Yaskawa INFORM job: X2_27-28(-50,-90).JBI

/JOB
//NAME X2_27-28(-50,-90)
//POS
///NPOS 352,352,352,16,0,0
///TOOL 0
///POSTYPE PULSE
///PULSE
C00000=-2348,-136985,-121477,-16,96092,-119
C00001=102627,-116827,-115343,23688,103226,-44542
C00002=115004,-86962,-92134,24001,100691,-40453
C00003=118842,-87386,-89376,23795,97842,-39618
C00004=120381,-87384,-88200,23717,96741,-39273
C00005=120377,-87274,-86494,23659,95829,-39457
C00006=120358,-87289,-86697,23665,95942,-39442
C00007=122537,-87238,-86673,23616,95334,-38762
C00008=120358,-87289,-86697,23665,95942,-39442
C00009=120413,-87366,-86683,23662,95882,-39433
C00010=120414,-83407,-84990,23721,96794,-39250
C00011=120413,-87366,-86683,23662,95882,-39433
C00012=118874,-87417,-87880,23731,96972,-39781
C00013=115033,-87126,-90695,23913,99792,-40627
C00014=115188,-84882,-91157,24044,101067,-40307
C00015=118973,-85347,-88418,23826,98226,-39491
C00016=120455,-85363,-87251,23745,97137,-39166
C00017=120452,-85286,-85558,23683,96217,-39352
C00018=120487,-85295,-85812,23691,96347,-39313
C00019=122635,-85238,-85785,23639,95749,-38643
C00020=120487,-85295,-85812,23691,96347,-39313
C00021=120483,-89746,-89095,23675,96102,-39363
C00022=120398,-93403,-88367,23560,93986,-39817
C00023=120400,-89378,-86736,23609,94965,-39621
C00024=120398,-93403,-88367,23560,93986,-39817
C00025=114754,-95185,-95401,23812,98729,-40947
C00026=113817,-96176,-94667,23309,84492,-38861
C00027=117813,-93582,-90807,22657,82424,-37804
C00028=119373,-92438,-89214,22393,81636,-37384
C00029=121634,-92435,-89210,21971,81030,-36673
C00030=120812,-92629,-89389,22126,81259,-36930
C00031=120809,-92377,-87626,22175,80372,-37096
C00032=120812,-92629,-89389,22126,81259,-36930
C00033=120909,-77641,-83091,21971,84792,-36245
C00034=120897,-73822,-81314,21956,85603,-36101
C00035=120909,-77641,-83091,21971,84792,-36245
C00036=115943,-80689,-88441,22878,87717,-37472
C00037=114304,-84462,-91699,24296,79100,-50020
C00038=117993,-82622,-88033,23316,76858,-49124
C00039=119438,-81769,-86512,22922,76000,-48762
C00040=121534,-81768,-86509,22277,75434,-48100
C00041=120893,-81605,-86471,22471,75662,-48293
C00042=120882,-79116,-84088,22491,75491,-48329
C00043=120893,-81605,-86471,22471,75662,-48293
C00044=120874,-97072,-87829,23296,69089,-49605
C00045=120882,-99825,-87797,23508,67765,-49878
C00046=120874,-97072,-87829,23296,69089,-49605
C00047=115137,-101258,-93439,24799,71949,-51221
C00048=121122,-106374,-107449,-1374,89824,-2285
C00049=126924,-83388,-91593,-24529,79629,49999
C00050=123244,-81641,-87969,-23551,77363,49118
C00051=121801,-80822,-86464,-23159,76497,48761
C00052=119718,-80838,-86473,-22519,75929,48107
C00053=120355,-80669,-86431,-22711,76157,48297
C00054=120355,-78205,-84050,-22728,75972,48332
C00055=120355,-80669,-86431,-22711,76157,48297
C00056=120389,-96242,-87887,-23521,69604,49623
C00057=120385,-99021,-87874,-23730,68282,49899
C00058=120389,-96242,-87887,-23521,69604,49623
C00059=126112,-100299,-93445,-25011,72503,51215
C00060=127424,-95125,-94496,-23537,84985,38865
C00061=123439,-92623,-90674,-22887,82890,37821
C00062=121881,-91514,-89094,-22623,82092,37406
C00063=119636,-91530,-89104,-22205,81483,36703
C00064=120453,-91715,-89278,-22359,81714,36957
C00065=120449,-91492,-87527,-22405,80819,37124
C00066=120453,-91715,-89278,-22359,81714,36957
C00067=120324,-76745,-82936,-22209,85198,36262
C00068=120328,-72933,-81149,-22194,85997,36116
C00069=120324,-76745,-82936,-22209,85198,36262
C00070=125282,-79685,-88237,-23118,88153,37475
C00071=126053,-84105,-90945,-24270,101400,40334
C00072=121317,-84665,-86997,-23961,97551,39378
C00073=120794,-84655,-86302,-23916,97014,39294
C00074=120791,-84616,-85408,-23898,96528,39392
C00075=120757,-84623,-85661,-23907,96658,39353
C00076=118619,-84583,-85646,-23856,96058,38687
C00077=120757,-84623,-85661,-23907,96658,39353
C00078=120851,-89642,-89189,-23884,96311,39457
C00079=120861,-92728,-88235,-23770,94318,39863
C00080=120850,-88708,-86596,-23821,95285,39665
C00081=120861,-92728,-88235,-23770,94318,39863
C00082=126087,-84100,-90943,-24271,101411,40344
C00083=126241,-86175,-91925,-24226,101032,40481
C00084=121422,-86671,-87791,-23936,97086,39512
C00085=120872,-86641,-86990,-23895,96491,39430
C00086=120871,-86598,-86346,-23873,96146,39499
C00087=120890,-86611,-86548,-23880,96260,39483
C00088=118722,-86577,-86536,-23832,95649,38808
C00089=120890,-86611,-86548,-23880,96260,39483
C00090=105063,-136064,-103329,-13656,63018,16453
C00091=105943,-129413,-101511,-13642,65401,16501
C00092=120836,-86689,-86535,-23876,96200,39475
C00093=126205,-86358,-90494,-24135,100129,40655
C00094=125851,-82973,-83923,-27955,66645,49280
C00095=122078,-79433,-79887,-26568,64829,48204
C00096=120947,-75344,-77359,-25987,64969,47712
C00097=120941,-87606,-78058,-27327,59684,49044
C00098=122175,-43746,-63261,-25567,94939,41852
C00099=109367,-31323,-61147,-11102,108854,34189
C00100=107960,-73866,-84355,-11763,95605,26787
C00101=120197,-78516,-82664,-23544,93398,30256
C00102=120674,-129805,-92807,-30414,50954,51524
C00103=120568,-142544,-87811,-37090,40465,55803
C00104=123719,-144899,-89705,-38330,41729,57027
C00105=131684,-150990,-93667,-41315,44633,60156
C00106=129569,-143343,-101170,-37382,56065,55166
C00107=120626,-84262,-98768,-23738,98439,36527
C00108=120626,-85138,-96217,-23600,96582,36901
C00109=120626,-85456,-94922,-23545,95698,37077
C00110=120469,-86348,-95216,-23512,95399,37081
C00111=120625,-86136,-87716,-24840,69295,42376
C00112=120625,-84905,-79807,-28619,54750,46053
C00113=120674,-84200,-73221,-29616,52346,46820
C00114=120694,-85495,-80856,-24885,69158,42438
C00115=120625,-86085,-86255,-23338,89936,38209
C00116=120426,-89896,-87913,-23311,89017,38317
C00117=120625,-86141,-87502,-23348,90617,38076
C00118=120625,-86117,-90396,-23390,92270,37753
C00119=121122,-106374,-107449,-1374,89824,-2285
C00120=115389,-83619,-83840,27729,66202,-49282
C00121=119161,-80016,-79774,26335,64406,-48194
C00122=120546,-78290,-78340,25753,63980,-47732
C00123=118816,-53732,-67922,25413,88359,-43218
C00124=120555,-20800,-48886,25341,110394,-38056
C00125=120540,-55987,-71055,24625,106356,-38968
C00126=122541,-110534,-92373,22580,69456,-43286
C00127=118405,-143902,-85879,49364,33417,-58427
C00128=117619,-149172,-81328,56749,30391,-62419
C00129=116407,-166632,-89102,63406,28902,-66105
C00130=115676,-54235,-75024,25023,110799,-39825
C00131=118805,-64147,-80292,27733,101935,-40879
C00132=120626,-85310,-99014,23481,98015,-36524
C00133=120626,-86187,-96453,23350,96148,-36894
C00134=120608,-87043,-95140,23285,95004,-37126
C00135=120561,-87834,-95469,23281,94829,-37179
C00136=120625,-86662,-87587,24592,68893,-42354
C00137=120624,-85616,-79792,28395,54313,-46043
C00138=120594,-85215,-73113,29470,51713,-46859
C00139=120625,-86330,-81078,24616,68777,-42377
C00140=119608,-72473,-79941,24560,98029,-43290
C00141=120456,-60135,-73698,25012,105696,-48505
C00142=120625,-87037,-87669,23119,90208,-38053
C00143=120626,-87011,-90570,23155,91868,-37731
C00144=120666,-77011,-108669,24508,106824,-34682
C00145=120666,-77011,-108669,24508,106824,-34682
C00146=69969,-70044,-127853,-26190,66176,42607
C00147=164066,-57873,-122395,-24689,68505,41679
C00148=164066,-57873,-122395,-24689,68505,41679
C00149=160176,-49519,-119791,-24551,119921,39872
C00150=160176,-63483,-121326,-22850,113002,41438
C00151=158640,-65340,-120741,-22195,111473,41297
C00152=158591,-68589,-120293,-21868,109653,41643
C00153=157443,-69457,-121106,-21570,109470,41332
C00154=156525,-70687,-121652,-21280,109008,41144
C00155=157421,-68776,-121134,-21620,109807,41260
C00156=165312,-86424,-128504,-22962,107296,44197
C00157=165830,-86354,-127308,-22986,106767,44469
C00158=165199,-83493,-126223,-22948,107364,44147
C00159=166594,-89849,-128602,-23030,106020,44865
C00160=164066,-57873,-122395,-24689,117052,41679
C00161=137183,-48540,-113103,-27062,110870,33097
C00162=133437,-50146,-110771,-25387,107987,32705
C00163=131981,-50551,-109735,-24766,106894,32528
C00164=131972,-53362,-109280,-24521,105318,32870
C00165=131636,-52132,-109559,-24518,105977,32629
C00166=130703,-53161,-109590,-24138,105304,32500
C00167=129879,-53398,-109717,-23857,105082,32305
C00168=131928,-52773,-109383,-24556,105642,32786
C00169=129764,-110950,-131053,-20350,81074,33499
C00170=129689,-122862,-131886,-20674,75787,34382
C00171=129370,-114001,-129067,-20345,78360,33827
C00172=129689,-122862,-131886,-20674,75787,34382
C00173=132778,-100905,-131254,-21387,86712,33498
C00174=143318,-75184,-130722,-7426,108145,5953
C00175=142042,-70835,-125479,-6985,107076,5675
C00176=141569,-69161,-123389,-6821,106623,5573
C00177=141558,-72780,-123049,-6738,104567,5686
C00178=141593,-72294,-123187,-6761,104902,5677
C00179=140967,-66354,-120569,-6623,106293,5428
C00180=141593,-72294,-123187,-6761,104902,5677
C00181=143345,-79213,-130741,-7340,106105,6087
C00182=143299,-74412,-130544,-7434,108429,5930
C00183=142026,-70178,-125329,-6991,107319,5656
C00184=141554,-68541,-123249,-6826,106852,5556
C00185=141544,-72173,-122918,-6742,104795,5669
C00186=141535,-71558,-123086,-6755,105212,5644
C00187=140912,-65651,-120469,-6618,106588,5397
C00188=141535,-71558,-123086,-6755,105212,5644
C00189=143280,-78289,-130595,-7337,106482,6046
C00190=143232,-73654,-130370,-7428,108704,5895
C00191=141965,-69530,-125182,-6983,107555,5626
C00192=141496,-67928,-123110,-6817,107076,5527
C00193=141485,-71574,-122787,-6732,105017,5641
C00194=141522,-70879,-122980,-6762,105492,5624
C00195=140900,-65004,-120364,-6625,106853,5379
C00196=141522,-70879,-122980,-6762,105492,5624
C00197=143263,-77436,-130447,-7347,106826,6020
C00198=97122,-37708,-107994,29413,114613,-34215
C00199=100765,-40257,-106178,27624,111617,-33971
C00200=102190,-41052,-105346,26964,110463,-33848
C00201=102184,-43828,-104954,26656,108968,-34218
C00202=102229,-43254,-105047,26705,109274,-34130
C00203=104151,-44223,-105589,26045,108681,-33706
C00204=102229,-43254,-105047,26705,109274,-34130
C00205=102390,-95092,-126215,23236,87986,-35228
C00206=102126,-106454,-127212,23433,83236,-36243
C00207=102723,-99043,-124596,23148,85111,-35678
C00208=102126,-106454,-127212,23433,83236,-36243
C00209=98351,-76946,-122874,24964,95636,-34932
C00210=98001,-57475,-123101,17996,113820,-36592
C00211=101536,-60773,-120906,16470,110382,-36160
C00212=102910,-63141,-119733,15828,108317,-36071
C00213=102916,-65026,-119479,15713,107233,-36217
C00214=102928,-64308,-119579,15751,107645,-36158
C00215=105169,-65555,-120144,15037,107042,-35610
C00216=102928,-64308,-119579,15751,107645,-36158
C00217=100368,-93898,-131351,15864,100368,-37874
C00218=97661,-87630,-128580,16731,102276,-38427
C00219=97996,-84252,-127310,16710,103135,-38207
C00220=97637,-87591,-128732,16747,102389,-38418
C00221=98001,-57475,-123101,17996,113820,-36592
C00222=99672,-7498,-88471,25376,120102,-35641
C00223=102088,-13346,-89114,23936,117260,-35660
C00224=103047,-14853,-89113,23458,116364,-35598
C00225=103070,-15280,-89318,23419,116275,-35613
C00226=103053,-14956,-89343,23464,116445,-35580
C00227=111428,-26181,-98637,10737,112296,-30408
C00228=102060,-12538,-89166,24052,117675,-35572
C00229=99645,-6651,-88487,25511,120511,-35544
C00230=110953,-13508,-91662,10573,109125,24437
C00231=110055,-18058,-91129,10746,106581,23991
C00232=118115,-24092,-94041,-1176,104714,22608
C00233=109847,-18561,-90498,10785,105963,23883
C00234=111445,-19708,-91242,10156,105696,24257
C00235=118682,-20843,-91970,7294,105023,25985
C00236=108853,-8664,-84384,24098,112429,23291
C00237=120831,-18883,-92219,6481,106051,26563
C00238=108247,-47697,-110693,11257,103619,23266
C00239=108001,-45758,-107370,11293,102615,23108
C00240=93743,-22704,-93084,31932,116237,9910
C00241=103043,-28379,-96833,28832,113378,11880
C00242=99567,-22662,-96038,30605,116358,11712
C00243=121744,-14004,-92551,6221,108699,26920
C00244=120102,-53038,-115079,-8947,92663,44391
C00245=120610,-122376,-128753,-45788,73253,81068
C00246=120610,-123649,-126232,-46257,71693,81820
C00247=114942,-121659,-128592,-38094,72140,80087
C00248=110746,-115512,-128718,-32121,74014,77680
C00249=111140,-116612,-128713,-32226,73312,78150
C00250=112123,-116971,-127920,-32543,72557,78927
C00251=114439,-125713,-130131,-33559,69229,81351
C00252=117557,-125023,-128034,-34922,66197,84237
C00253=123831,-113405,-131509,-37414,82436,80766
C00254=120611,-116611,-133297,-36284,80720,80097
C00255=120611,-116611,-133297,-36284,54343,80097
C00256=99428,-107843,-133398,6584,68498,81557
C00257=78879,-54177,-103402,55937,89044,85268
C00258=78429,-99723,-127104,45672,96643,84222
C00259=82364,-110385,-127773,44232,91185,83459
C00260=83904,-116944,-128983,43779,88549,82984
C00261=84962,-116458,-129077,42971,88317,83920
C00262=85753,-115873,-128369,42851,86976,84102
C00263=94278,-102678,-129331,33632,95313,84379
C00264=94252,-98051,-127422,33733,96332,84676
C00265=92227,-97102,-128188,34391,97842,84417
C00266=83296,-105916,-131418,40048,95342,83077
C00267=112976,-81346,-133029,11053,104292,84731
C00268=138914,-76030,-130615,-14013,102422,84743
C00269=139405,-82424,-128484,-14961,97637,85019
C00270=139610,-84860,-127656,-14962,95960,85285
C00271=122825,-93017,-130267,6502,91067,84006
C00272=122185,-92165,-130257,6747,91537,83850
C00273=122216,-90116,-129760,6745,92278,83897
C00274=121098,-81728,-131688,7259,97815,83901
C00275=117564,-73996,-132555,6245,103794,67045
C00276=120619,-75058,-128623,-5257,106122,114
C00277=120619,-82255,-128190,-5150,102172,284
C00278=120619,-84669,-127718,-5117,100646,349
C00279=112025,-83330,-127195,-2462,100682,-2074
C00280=125410,-84211,-127707,-6591,101158,1679
C00281=116389,-83882,-127652,-3819,100819,-855
C00282=120619,-81538,-128040,-5156,102448,272
C00283=120619,-74311,-128456,-5266,106402,102
C00284=120619,-74726,-128566,4732,106271,-192
C00285=120619,-81960,-128145,4635,102308,-346
C00286=120619,-84896,-127978,4605,100704,-408
C00287=130171,-82621,-126955,1656,100942,2285
C00288=124481,-84935,-127680,3411,100342,674
C00289=124544,-84819,-127737,3393,100431,696
C00290=120619,-82679,-128294,4629,102031,-356
C00291=132569,-75475,-129249,4725,105990,-203
C00292=136339,-73848,-128583,3524,106271,812
C00293=115610,-90997,-132796,9664,98154,47330
C00294=101030,-93647,-129382,39129,95529,59479
C00295=126122,-118259,-133558,37742,75798,85079
C00296=126123,-123502,-128947,38676,71399,83468
C00297=126367,-125496,-128832,38806,70431,83204
C00298=126259,-125638,-129343,38123,70704,84047
C00299=126452,-122750,-128309,37875,71302,84347
C00300=126394,-120456,-127460,37773,71850,84523
C00301=124054,-126150,-130879,35007,72357,80836
C00302=128390,-137176,-133704,31743,64167,79569
C00303=127393,-110720,-125425,30503,71855,81401
C00304=124670,-119490,-131862,32313,77272,81796
C00305=123468,-105545,-131306,32649,85926,83785
C00306=123468,-105545,-131306,32649,65045,83785
C00307=138629,-76986,-116006,-44057,63514,71452
C00308=138629,-76986,-116006,-43820,94287,71434
C00309=134687,-82864,-115400,-42250,90109,71636
C00310=135664,-119265,-122373,-47079,71549,79745
C00311=132914,-91853,-117066,-41458,84473,72364
C00312=132788,-89730,-116313,-41385,84897,72145
C00313=132694,-88516,-115506,-41345,84954,72084
C00314=132043,-80417,-112459,-40576,87939,70586
C00315=130204,-77793,-113758,-38013,92059,70441
C00316=128524,-79115,-118595,-35047,97544,70713
C00317=132051,-72530,-119355,-36693,101910,70485
C00318=103939,-76664,-132684,-5369,102917,72052
C00319=89328,-90531,-135287,12506,96574,73027
C00320=80068,-79251,-126452,22073,101797,73002
C00321=79731,-82396,-126595,22049,100450,72647
C00322=75389,-93321,-128367,26734,94516,71144
C00323=89823,-118490,-137568,8328,79761,70288
C00324=89823,-118490,-137568,8328,79761,70288
C00325=89554,-115143,-136518,8419,80849,70278
C00326=90481,-87040,-133249,3898,95478,71874
C00327=121995,-40580,-113920,-16331,113160,53817
C00328=134131,-13261,-91828,-23304,117904,34003
C00329=134130,-17922,-91482,-22725,115495,34532
C00330=134178,-18161,-90930,-22645,115075,34636
C00331=134130,-19018,-91366,-22584,114907,34660
C00332=134135,-19080,-91406,-22584,114899,34666
C00333=130040,-16797,-91734,-17058,116519,30349
C00334=134130,-17121,-91555,-22821,115917,34441
C00335=134485,-13609,-94717,-23816,119438,33744
C00336=134125,-15266,-91655,-12564,108610,-23590
C00337=134126,-19967,-91222,-12356,105989,-23311
C00338=128619,-18785,-91351,-4606,108870,-22773
C00339=134001,-21196,-91423,-12272,105476,-23287
C00340=133837,-21232,-91027,-12191,105205,-23306
C00341=133810,-21099,-91074,-12188,105299,-23320
C00342=142675,1303,-75956,-28153,117136,-18516
C00343=136270,-18169,-92488,-13326,107877,-22987
C00344=160414,-17591,-92076,-34517,119430,-9586
C00345=156591,-5353,-82577,-31368,124461,-10572
C00346=145789,-11555,-87834,-25790,123238,-6673
C00347=150771,-16897,-91755,-28044,119951,-5168
C00348=137962,-9823,-90715,-14308,111174,-22977
C00349=135096,-37202,-106359,-15392,53710,-23809
C00350=91634,-70237,-111781,-11635,26322,-15777
C00351=-2394,-140510,-122466,-18,94889,-134
BC00000=133244,518772,1075139
BC00001=133244,374008,1075139
BC00002=133244,374008,1075139
BC00003=133244,374008,1075139
BC00004=133244,374008,1075139
BC00005=133244,374008,1075139
BC00006=133244,374008,1075139
BC00007=133244,374008,1075139
BC00008=133244,374008,1075139
BC00009=133244,374008,1075139
BC00010=133244,374008,1075139
BC00011=133244,374008,1075139
BC00012=133244,374008,1075139
BC00013=133244,374008,1075139
BC00014=133336,405551,1075139
BC00015=133336,405551,1075139
BC00016=133336,405551,1075139
BC00017=133336,405551,1075139
BC00018=133336,405551,1075139
BC00019=133336,405551,1075139
BC00020=133336,405551,1075139
BC00021=133336,405551,1075139
BC00022=133336,405551,1075139
BC00023=133336,405551,1075139
BC00024=133336,405551,1075139
BC00025=133336,405551,1075139
BC00026=104477,408619,1075139
BC00027=104477,408619,1075139
BC00028=104477,408619,1075139
BC00029=104477,408619,1075139
BC00030=104477,408619,1075139
BC00031=104477,408619,1075139
BC00032=104477,408619,1075139
BC00033=104477,408619,1075139
BC00034=104477,408619,1075139
BC00035=104477,408619,1075139
BC00036=104477,408619,1075139
BC00037=104582,411051,1075139
BC00038=104582,411051,1075139
BC00039=104582,411051,1075139
BC00040=104582,411051,1075139
BC00041=104582,411051,1075139
BC00042=104582,411051,1075139
BC00043=104582,411051,1075139
BC00044=104582,411051,1075139
BC00045=104582,411051,1075139
BC00046=104582,411051,1075139
BC00047=104582,411051,1075139
BC00048=209905,391148,1075139
BC00049=330495,411073,1075139
BC00050=330495,411073,1075139
BC00051=330495,411073,1075139
BC00052=330495,411073,1075139
BC00053=330495,411073,1075139
BC00054=330495,411073,1075139
BC00055=330495,411073,1075139
BC00056=330495,411073,1075139
BC00057=330495,411073,1075139
BC00058=330495,411073,1075139
BC00059=330495,411073,1075139
BC00060=330336,408559,1075139
BC00061=330336,408559,1075139
BC00062=330336,408559,1075139
BC00063=330336,408559,1075139
BC00064=330336,408559,1075139
BC00065=330336,408559,1075139
BC00066=330336,408559,1075139
BC00067=330336,408559,1075139
BC00068=330336,408559,1075139
BC00069=330336,408559,1075139
BC00070=330336,408559,1075139
BC00071=301636,405299,1075139
BC00072=301637,405300,1075138
BC00073=301637,405300,1075137
BC00074=301636,405299,1075139
BC00075=301636,405299,1075139
BC00076=301636,405299,1075139
BC00077=301636,405299,1075139
BC00078=301636,405299,1075139
BC00079=301636,405299,1075139
BC00080=301636,405299,1075139
BC00081=301636,405299,1075139
BC00082=301636,405299,1075139
BC00083=301924,373758,1075139
BC00084=301924,373758,1075139
BC00085=301924,373758,1075139
BC00086=301924,373758,1075139
BC00087=301924,373758,1075139
BC00088=301924,373758,1075139
BC00089=301924,373758,1075139
BC00090=301924,373758,1075139
BC00091=301924,373758,1075139
BC00092=301924,373758,1075139
BC00093=301924,373758,1075139
BC00094=304905,422275,1075139
BC00095=304905,422275,1075139
BC00096=304905,422275,1075139
BC00097=304905,422275,1075139
BC00098=304905,422275,1075139
BC00099=304905,422275,1075139
BC00100=304905,422275,1075139
BC00101=304905,422275,1075139
BC00102=304905,422275,1075139
BC00103=304905,422275,1075139
BC00104=304905,422275,1075139
BC00105=304905,422275,1075139
BC00106=308182,411224,1075150
BC00107=321948,364809,1075193
BC00108=327549,363919,1075193
BC00109=329789,363562,1075193
BC00110=329784,365099,1075193
BC00111=329679,406352,1075193
BC00112=329645,424796,1075193
BC00113=329621,438429,1075193
BC00114=329656,420343,1075193
BC00115=329731,391181,1075193
BC00116=329680,407690,1075193
BC00117=327439,408070,1075193
BC00118=321838,409018,1075193
BC00119=209905,391148,1075139
BC00120=130051,422412,1075139
BC00121=130051,422412,1075139
BC00122=130051,422412,1075139
BC00123=130051,422412,1075139
BC00124=130051,422412,1075139
BC00125=130051,422412,1075139
BC00126=130051,422412,1075139
BC00127=130051,422412,1075139
BC00128=130052,422412,1075139
BC00129=130051,422412,1075139
BC00130=130051,422412,1075139
BC00131=129375,420117,1075141
BC00132=113133,364939,1075193
BC00133=107556,364016,1075193
BC00134=105325,363648,1075192
BC00135=105320,365183,1075193
BC00136=105215,406346,1075193
BC00137=105181,424701,1075193
BC00138=105157,438341,1075193
BC00139=105192,420360,1075193
BC00140=105266,391265,1075193
BC00141=105215,407774,1075193
BC00142=107446,408166,1075193
BC00143=113024,409146,1075193
BC00144=113024,409146,1075193
BC00145=113024,615302,1075193
BC00146=61085,522072,1075139
BC00147=61085,522072,1075139
BC00148=61085,344205,1075139
BC00149=61085,344205,1072934
BC00150=61085,344205,1075139
BC00151=61085,344205,1075139
BC00152=61085,344205,1075139
BC00153=61085,344205,1075139
BC00154=61085,344205,1075139
BC00155=61085,344205,1075139
BC00156=61085,344205,1075139
BC00157=61085,344205,1075139
BC00158=61085,344205,1075139
BC00159=61085,344205,1075139
BC00160=61085,344205,1075139
BC00161=23280,347448,1075139
BC00162=23280,347448,1075139
BC00163=23280,347448,1075139
BC00164=23280,347448,1075139
BC00165=23280,347448,1075139
BC00166=23280,347448,1075139
BC00167=23280,347448,1075139
BC00168=23280,347448,1075139
BC00169=23280,347448,1075139
BC00170=23280,347448,1075139
BC00171=23280,347448,1075139
BC00172=23280,347448,1075139
BC00173=23280,347448,1075139
BC00174=188977,346610,1075139
BC00175=188977,346610,1075139
BC00176=188977,346610,1075139
BC00177=188977,346610,1075139
BC00178=188977,346610,1075139
BC00179=188977,346610,1075139
BC00180=188977,346610,1075139
BC00181=188977,346610,1075139
BC00182=244494,346740,1075139
BC00183=244494,346740,1075139
BC00184=244494,346740,1075139
BC00185=244494,346740,1075139
BC00186=244494,346740,1075139
BC00187=244494,346740,1075139
BC00188=244494,346740,1075139
BC00189=244494,346740,1075139
BC00190=299376,346854,1075139
BC00191=299376,346854,1075139
BC00192=299376,346854,1075139
BC00193=299376,346854,1075139
BC00194=299376,346854,1075139
BC00195=299376,346854,1075139
BC00196=299376,346854,1075139
BC00197=299376,346854,1075139
BC00198=398158,351394,1075139
BC00199=398158,351394,1075139
BC00200=398158,351394,1075139
BC00201=398158,351394,1075139
BC00202=398158,351394,1075139
BC00203=398158,351394,1075139
BC00204=398158,351394,1075139
BC00205=398158,351394,1075139
BC00206=398158,351394,1075139
BC00207=398158,351394,1075139
BC00208=398158,351394,1075139
BC00209=398158,351394,1075139
BC00210=398158,355332,1075139
BC00211=398158,355332,1075139
BC00212=398158,355332,1075139
BC00213=398158,355332,1075139
BC00214=398158,355332,1075139
BC00215=398158,355332,1075139
BC00216=398158,355332,1075139
BC00217=398158,355332,1075139
BC00218=398158,355332,1075139
BC00219=398158,355332,1075139
BC00220=398158,355332,1075139
BC00221=398158,355332,1075139
BC00222=398158,400322,1075139
BC00223=398158,397462,1075139
BC00224=398158,396318,1075139
BC00225=398158,391714,1075139
BC00226=398158,377425,1075139
BC00227=398158,372820,1075139
BC00228=398158,373964,1075139
BC00229=398158,376823,1075139
BC00230=398158,418089,1075139
BC00231=398158,413055,1075139
BC00232=398158,411041,1075139
BC00233=398158,411041,1075139
BC00234=398158,407701,1075139
BC00235=398158,394074,1075139
BC00236=398157,390799,1075138
BC00237=398158,392757,1075139
BC00238=398158,392757,1075139
BC00239=398158,392757,1075139
BC00240=398158,392757,1075139
BC00241=398158,392757,1075139
BC00242=398158,392757,1075139
BC00243=398158,397791,1075139
BC00244=368036,376425,1075139
BC00245=305380,328053,1075139
BC00246=311014,327368,1075139
BC00247=313268,327093,1075139
BC00248=314020,306251,1075134
BC00249=314937,305830,1075134
BC00250=316315,305197,1075135
BC00251=320257,303387,1075136
BC00252=325137,301146,1075137
BC00253=323904,301076,1075139
BC00254=319263,301619,1075139
BC00255=319263,301619,1075139
BC00256=354630,317867,1075139
BC00257=398158,344123,1075139
BC00258=398158,328829,1075139
BC00259=398158,328117,1075139
BC00260=398158,327832,1075139
BC00261=398158,306302,1075139
BC00262=398158,307654,1075139
BC00263=398158,299863,1075139
BC00264=398158,299863,1075139
BC00265=398158,299850,1075139
BC00266=398158,299818,1075139
BC00267=398158,306594,1075139
BC00268=398158,312941,1075139
BC00269=398158,312327,1075139
BC00270=398158,311910,1075139
BC00271=398158,311948,1075139
BC00272=398158,311948,1075139
BC00273=398158,311948,1075139
BC00274=398158,312262,1075139
BC00275=361275,323313,1075139
BC00276=206057,349327,1075139
BC00277=206787,343889,1075139
BC00278=207078,341714,1075139
BC00279=207078,341714,1075139
BC00280=265248,341851,1075139
BC00281=265248,341851,1075139
BC00282=264956,344026,1075139
BC00283=264226,349464,1075139
BC00284=226795,349421,1075139
BC00285=226137,343980,1075139
BC00286=225873,341804,1075139
BC00287=225873,341804,1075139
BC00288=182394,341701,1075139
BC00289=167704,341666,1075139
BC00290=167967,343843,1075139
BC00291=168625,349284,1075139
BC00292=168625,349284,1075139
BC00293=110827,349284,1075139
BC00294=117018,341898,1075139
BC00295=129083,327506,1075139
BC00296=123497,326795,1075139
BC00297=121263,326510,1075139
BC00298=120594,305154,1075139
BC00299=120594,305154,1075139
BC00300=120594,305154,1075139
BC00301=111835,301464,1075139
BC00302=111835,301467,1075137
BC00303=111835,301467,1075137
BC00304=111094,300785,1075138
BC00305=115319,301016,1075139
BC00306=115319,315076,1075139
BC00307=1592,364988,1075139
BC00308=1592,342862,1075139
BC00309=1592,342176,1075139
BC00310=1592,341902,1075139
BC00311=1592,321468,1075139
BC00312=1592,321468,1075139
BC00313=1592,321468,1075139
BC00314=1592,322137,1075139
BC00315=1592,315667,1075139
BC00316=1592,307060,1075139
BC00317=1592,307005,1075139
BC00318=5534,309480,1075139
BC00319=11068,305519,1075139
BC00320=9993,304471,1075139
BC00321=9607,304094,1075139
BC00322=9607,304094,1075139
BC00323=9607,304094,1075139
BC00324=9607,304094,1075139
BC00325=9607,304094,1075139
BC00326=1592,304326,1075139
BC00327=7124,350617,1075139
BC00328=20477,398593,1075139
BC00329=25318,395756,1075139
BC00330=27254,394622,1075139
BC00331=27284,390018,1075139
BC00332=27318,375728,1075139
BC00333=27313,372783,1075139
BC00334=25374,372258,1075139
BC00335=20533,375095,1075139
BC00336=41909,417655,1075139
BC00337=40292,412613,1075139
BC00338=39645,410596,1075139
BC00339=39645,410596,1075139
BC00340=42951,407272,1075139
BC00341=56475,393709,1075139
BC00342=56475,393709,1075139
BC00343=60436,392410,1075139
BC00344=60436,392410,1075139
BC00345=60435,392411,1075136
BC00346=60435,392411,1075136
BC00347=60435,392411,1075136
BC00348=62053,397452,1075139
BC00349=63646,397452,1075139
BC00350=86333,436115,1075139
BC00351=134837,518772,1075139
EC00000=443420,372643
EC00001=443420,372643
EC00002=443420,372643
EC00003=443420,372643
EC00004=443420,372643
EC00005=443420,372643
EC00006=443420,372643
EC00007=443420,372643
EC00008=443420,372643
EC00009=443420,372643
EC00010=443420,372643
EC00011=443420,372643
EC00012=443420,372643
EC00013=443420,372643
EC00014=443420,372643
EC00015=443420,372643
EC00016=443420,372643
EC00017=443420,372643
EC00018=443420,372643
EC00019=443420,372643
EC00020=443420,372643
EC00021=443420,372643
EC00022=443420,372643
EC00023=443420,372643
EC00024=443420,372643
EC00025=443420,372643
EC00026=443420,372643
EC00027=443420,372643
EC00028=443420,372643
EC00029=443420,372643
EC00030=443420,372643
EC00031=443420,372643
EC00032=443420,372643
EC00033=443420,372643
EC00034=443420,372643
EC00035=443420,372643
EC00036=443420,372643
EC00037=443420,372643
EC00038=443420,372643
EC00039=443420,372643
EC00040=443420,372643
EC00041=443420,372643
EC00042=443420,372643
EC00043=443420,372643
EC00044=443420,372643
EC00045=443420,372643
EC00046=443420,372643
EC00047=443420,372643
EC00048=443420,372643
EC00049=443420,372643
EC00050=443420,372643
EC00051=443420,372643
EC00052=443420,372643
EC00053=443420,372643
EC00054=443420,372643
EC00055=443420,372643
EC00056=443420,372643
EC00057=443420,372643
EC00058=443420,372643
EC00059=443420,372643
EC00060=443420,372643
EC00061=443420,372643
EC00062=443420,372643
EC00063=443420,372643
EC00064=443420,372643
EC00065=443420,372643
EC00066=443420,372643
EC00067=443420,372643
EC00068=443420,372643
EC00069=443420,372643
EC00070=443420,372643
EC00071=443420,372643
EC00072=443419,372644
EC00073=443418,372644
EC00074=443420,372643
EC00075=443420,372643
EC00076=443420,372643
EC00077=443420,372643
EC00078=443420,372643
EC00079=443420,372643
EC00080=443420,372643
EC00081=443420,372643
EC00082=443420,372643
EC00083=443420,372643
EC00084=443420,372643
EC00085=443420,372643
EC00086=443420,372643
EC00087=443420,372643
EC00088=443420,372643
EC00089=443420,372643
EC00090=443420,372643
EC00091=443420,372643
EC00092=443420,372643
EC00093=443420,372643
EC00094=443420,372643
EC00095=443420,372643
EC00096=443420,372643
EC00097=443420,372643
EC00098=443420,372643
EC00099=443420,372643
EC00100=443420,372643
EC00101=443420,372643
EC00102=443420,372643
EC00103=443420,372643
EC00104=443420,372643
EC00105=443420,372643
EC00106=443420,372643
EC00107=443420,372643
EC00108=443420,372643
EC00109=443420,372643
EC00110=443420,372643
EC00111=443420,372643
EC00112=443420,372643
EC00113=443420,372643
EC00114=443420,372643
EC00115=443420,372643
EC00116=443420,372643
EC00117=443420,372643
EC00118=443420,372643
EC00119=443420,372643
EC00120=443420,372643
EC00121=443420,372643
EC00122=443420,372643
EC00123=443420,372643
EC00124=443420,372643
EC00125=443420,372643
EC00126=443420,372643
EC00127=443420,372643
EC00128=443419,372642
EC00129=443420,372643
EC00130=443420,372643
EC00131=443420,372643
EC00132=443420,372643
EC00133=443420,372643
EC00134=443419,372643
EC00135=443420,372643
EC00136=443420,372643
EC00137=443420,372643
EC00138=443420,372643
EC00139=443420,372643
EC00140=443420,372643
EC00141=443420,372643
EC00142=443420,372643
EC00143=443420,372643
EC00144=443420,372643
EC00145=443420,372643
EC00146=798156,372643
EC00147=798156,372643
EC00148=798156,372643
EC00149=798156,372643
EC00150=798156,372643
EC00151=798156,372643
EC00152=798156,372643
EC00153=798156,372643
EC00154=798156,372643
EC00155=798156,372643
EC00156=798156,372643
EC00157=798156,372643
EC00158=798156,372643
EC00159=798156,372643
EC00160=798156,372643
EC00161=798156,372643
EC00162=798156,372643
EC00163=798156,372643
EC00164=798156,372643
EC00165=798156,372643
EC00166=798156,372643
EC00167=798156,372643
EC00168=798156,372643
EC00169=798156,372643
EC00170=798156,372643
EC00171=798156,372643
EC00172=798156,372643
EC00173=798156,372643
EC00174=798156,372643
EC00175=798156,372643
EC00176=798156,372643
EC00177=798156,372643
EC00178=798156,372643
EC00179=798156,372643
EC00180=798156,372643
EC00181=798156,372643
EC00182=798156,372643
EC00183=798156,372643
EC00184=798156,372643
EC00185=798156,372643
EC00186=798156,372643
EC00187=798156,372643
EC00188=798156,372643
EC00189=798156,372643
EC00190=798156,372643
EC00191=798156,372643
EC00192=798156,372643
EC00193=798156,372643
EC00194=798156,372643
EC00195=798156,372643
EC00196=798156,372643
EC00197=798156,372643
EC00198=798156,372643
EC00199=798156,372643
EC00200=798156,372643
EC00201=798156,372643
EC00202=798156,372643
EC00203=798156,372643
EC00204=798156,372643
EC00205=798156,372643
EC00206=798156,372643
EC00207=798156,372643
EC00208=798156,372643
EC00209=798156,372643
EC00210=798156,372643
EC00211=798156,372643
EC00212=798156,372643
EC00213=798156,372643
EC00214=798156,372643
EC00215=798156,372643
EC00216=798156,372643
EC00217=798156,372643
EC00218=798156,372643
EC00219=798156,372643
EC00220=798156,372643
EC00221=798156,372643
EC00222=798156,372643
EC00223=798156,372643
EC00224=798156,372643
EC00225=798156,372643
EC00226=798156,372643
EC00227=798156,372643
EC00228=798156,372643
EC00229=798156,372643
EC00230=798156,372643
EC00231=798156,372643
EC00232=798156,372643
EC00233=798156,372643
EC00234=798156,372643
EC00235=798156,372643
EC00236=798153,372643
EC00237=798156,372643
EC00238=798156,372643
EC00239=798156,372643
EC00240=798156,372643
EC00241=798156,372643
EC00242=798156,372643
EC00243=798156,372643
EC00244=798156,372643
EC00245=798156,372643
EC00246=798156,372643
EC00247=798156,372643
EC00248=798154,372643
EC00249=798154,372643
EC00250=798155,372644
EC00251=798155,372644
EC00252=798155,372643
EC00253=798156,372643
EC00254=798156,372643
EC00255=798156,372643
EC00256=798156,372643
EC00257=798156,372643
EC00258=798156,372643
EC00259=798156,372643
EC00260=798156,372643
EC00261=798156,372643
EC00262=798156,372643
EC00263=798156,372643
EC00264=798156,372643
EC00265=798156,372643
EC00266=798156,372643
EC00267=798156,372643
EC00268=798156,372643
EC00269=798156,372643
EC00270=798156,372643
EC00271=798156,372643
EC00272=798156,372643
EC00273=798156,372643
EC00274=798156,372643
EC00275=798156,372643
EC00276=798156,372643
EC00277=798156,372643
EC00278=798156,372643
EC00279=798156,372643
EC00280=798156,372643
EC00281=798156,372643
EC00282=798156,372643
EC00283=798156,372643
EC00284=798156,372643
EC00285=798156,372643
EC00286=798156,372643
EC00287=798156,372643
EC00288=798156,372643
EC00289=798156,372643
EC00290=798156,372643
EC00291=798156,372643
EC00292=798156,372643
EC00293=798156,372643
EC00294=798156,372643
EC00295=798156,372643
EC00296=798156,372643
EC00297=798156,372643
EC00298=798156,372643
EC00299=798156,372643
EC00300=798156,372643
EC00301=798156,372643
EC00302=798155,372643
EC00303=798155,372643
EC00304=798156,372643
EC00305=798156,372643
EC00306=798156,372643
EC00307=798156,372643
EC00308=798156,372643
EC00309=798156,372643
EC00310=798156,372643
EC00311=798156,372643
EC00312=798156,372643
EC00313=798156,372643
EC00314=798156,372643
EC00315=798156,372643
EC00316=798156,372643
EC00317=798156,372643
EC00318=798156,372643
EC00319=798156,372643
EC00320=798156,372643
EC00321=798156,372643
EC00322=798156,372643
EC00323=798156,372643
EC00324=798156,372643
EC00325=798156,372643
EC00326=798156,372643
EC00327=798156,372643
EC00328=798156,372643
EC00329=798156,372643
EC00330=798156,372643
EC00331=798156,372643
EC00332=798156,372643
EC00333=798156,372643
EC00334=798156,372643
EC00335=798156,372643
EC00336=798156,372643
EC00337=798156,372643
EC00338=798156,372643
EC00339=798156,372643
EC00340=798156,372643
EC00341=798156,372643
EC00342=798156,372643
EC00343=798156,372643
EC00344=798156,372643
EC00345=798154,372643
EC00346=798154,372643
EC00347=798154,372643
EC00348=798156,372643
EC00349=798156,372643
EC00350=798156,372643
EC00351=798156,372643
///POSTYPE BASE
///RECTAN
///RCONF 0,0,0,0,1,0,0,0,0,0,0,0,0,0,0,0,0,0,0,0,0,0,0,0
P00006=2.006,1.622,-0.565,0.0000,0.0000,0.0000
P00021=0.073,2.058,-0.109,0.0000,0.0000,0.0000
P00022=2.006,1.622,-0.565,0.0000,0.0000,0.0000
///RCONF 0,0,0,0,0,0,0,0,0,0,0,0,0,0,0,0,0,0,0,0,0,0,0,0
P00023=-2.957,-4.083,2.762,0.0000,0.0000,0.0000
P00024=-1.466,-0.226,-0.419,0.0000,0.0000,0.0000
P00025=3.643,0.007,-2.585,0.0000,0.0000,0.0000
P00031=-0.170,0.039,-0.647,0.0000,0.0000,0.0000
P00032=-0.423,0.157,3.222,0.0000,0.0000,0.0000
P00033=0.854,-1.099,3.047,0.0000,0.0000,0.0000
///RCONF 0,0,0,0,1,0,0,0,0,0,0,0,0,0,0,0,0,0,0,0,0,0,0,0
P00034=-8.151,9.743,-4.393,0.0000,0.0000,0.0000
///RCONF 0,0,0,0,0,0,0,0,0,0,0,0,0,0,0,0,0,0,0,0,0,0,0,0
P00035=0.390,-0.027,1.040,0.0000,0.0000,0.0000
P00036=-2.434,0.084,0.197,0.0000,0.0000,0.0000
P00037=-1.075,5.090,-3.949,0.0000,0.0000,0.0000
P00038=0.174,-1.527,-10.860,0.0000,0.0000,0.0000
P00039=-0.109,1.838,-0.266,0.0000,0.0000,0.0000
P00040=2.716,-0.016,3.014,0.0000,0.0000,0.0000
//INST
///DATE 2024/12/18 15:24
///ATTR SC,RW
///GROUP1 RB1,BS1
///GROUP2 ST1
NOP
'X2_27-28(-50,-90)
'spoiny do polaczenia
MOVJ C00000 BC00000 VJ=100.00  +MOVJ EC00000 VJ=100.00
MOVJ C00001 BC00001 VJ=100.00  +MOVJ EC00001 VJ=100.00
'Path S4320
SSFTOF
SFTOF3D
MOVJ C00002 BC00002 VJ=100.00  +MOVJ EC00002 VJ=100.00
MOVL C00003 BC00003 V=800.0  +MOVJ EC00003 VJ=100.00
SMOVL C00004 BC00004 V=166.7  +MOVJ EC00004
SREFP 3 C00005 BC00005  +REFP EC00005
CALL JOB:SEARCH-R1-S13D
SET P033 P006
SFTON3D P033
SMOVL C00006 BC00006 V=166.7  +MOVJ EC00006
SREFP 3 C00007 BC00007  +REFP EC00007
CALL JOB:SEARCH-R1-S13D
SET P033 P006
SFTON3D P033
SMOVL C00008 BC00008 V=166.7  +MOVJ EC00008
SMOVL C00009 BC00009 V=166.7  +MOVJ EC00009
SREFP 3 C00010 BC00010  +REFP EC00010
CALL JOB:SEARCH-R1-S13D
SET P033 P006
SFTON3D P033
SMOVL C00011 BC00011 V=166.7  +MOVJ EC00011
MOVL C00012 BC00012 V=800.0  +MOVJ EC00012 VJ=100.00
MOVL C00013 BC00013 V=1000.0  +MOVJ EC00013 VJ=100.00
'EndPath S4320
'Path S4321
SFTOF3D
MOVJ C00014 BC00014 VJ=100.00  +MOVJ EC00014 VJ=100.00
MOVL C00015 BC00015 V=800.0  +MOVJ EC00015 VJ=100.00
SMOVL C00016 BC00016 V=166.7  +MOVJ EC00016
SREFP 3 C00017 BC00017  +REFP EC00017
CALL JOB:SEARCH-R1-S13D
SET P034 P006
SFTON3D P034
SMOVL C00018 BC00018 V=166.7  +MOVJ EC00018
SREFP 3 C00019 BC00019  +REFP EC00019
CALL JOB:SEARCH-R1-S13D
SET P034 P006
SFTON3D P034
SMOVL C00020 BC00020 V=166.7  +MOVJ EC00020
SMOVL C00021 BC00021 V=250.0  +MOVJ EC00021
SMOVL C00022 BC00022 V=166.7  +MOVJ EC00022
SREFP 3 C00023 BC00023  +REFP EC00023
CALL JOB:SEARCH-R1-S13D
SET P034 P006
SFTON3D P034
SMOVL C00024 BC00024 V=166.7  +MOVJ EC00024
MOVL C00025 BC00025 V=1000.0  +MOVJ EC00025 VJ=100.00
'EndPath S4321
'Path S4322
SFTOF3D
MOVJ C00026 BC00026 VJ=100.00  +MOVJ EC00026 VJ=100.00
MOVL C00027 BC00027 V=800.0  +MOVJ EC00027 VJ=100.00
SMOVL C00028 BC00028 V=166.7  +MOVJ EC00028
SREFP 3 C00029 BC00029  +REFP EC00029
CALL JOB:SEARCH-R1-S13D
SET P035 P006
SFTON3D P035
SMOVL C00030 BC00030 V=166.7  +MOVJ EC00030
SREFP 3 C00031 BC00031  +REFP EC00031
CALL JOB:SEARCH-R1-S13D
SET P035 P006
SFTON3D P035
SMOVL C00032 BC00032 V=166.7  +MOVJ EC00032
SMOVL C00033 BC00033 V=250.0  +MOVJ EC00033
SREFP 3 C00034 BC00034  +REFP EC00034
CALL JOB:SEARCH-R1-S13D
SET P035 P006
SFTON3D P035
SMOVL C00035 BC00035 V=250.0  +MOVJ EC00035
MOVL C00036 BC00036 V=1000.0  +MOVJ EC00036 VJ=100.00
'EndPath S4322
'Path S4323
SFTOF3D
MOVJ C00037 BC00037 VJ=100.00  +MOVJ EC00037 VJ=100.00
MOVL C00038 BC00038 V=800.0  +MOVJ EC00038 VJ=100.00
SMOVL C00039 BC00039 V=166.7  +MOVJ EC00039
SREFP 3 C00040 BC00040  +REFP EC00040
CALL JOB:SEARCH-R1-S13D
SET P036 P006
SFTON3D P036
SMOVL C00041 BC00041 V=166.7  +MOVJ EC00041
SREFP 3 C00042 BC00042  +REFP EC00042
CALL JOB:SEARCH-R1-S13D
SET P036 P006
SFTON3D P036
SMOVL C00043 BC00043 V=166.7  +MOVJ EC00043
SMOVL C00044 BC00044 V=250.0  +MOVJ EC00044
SREFP 3 C00045 BC00045  +REFP EC00045
CALL JOB:SEARCH-R1-S13D
SET P036 P006
SFTON3D P036
SMOVL C00046 BC00046 V=250.0  +MOVJ EC00046
MOVL C00047 BC00047 V=1000.0  +MOVJ EC00047 VJ=100.00
'EndPath S4323
'
MOVJ C00048 BC00048 VJ=100.00  +MOVJ EC00048 VJ=100.00
'Path S4328
SFTOF3D
MOVJ C00049 BC00049 VJ=100.00  +MOVJ EC00049 VJ=100.00
MOVL C00050 BC00050 V=800.0  +MOVJ EC00050 VJ=100.00
SMOVL C00051 BC00051 V=166.7  +MOVJ EC00051
SREFP 3 C00052 BC00052  +REFP EC00052
CALL JOB:SEARCH-R1-S13D
SET P040 P006
SFTON3D P040
SMOVL C00053 BC00053 V=166.7  +MOVJ EC00053
SREFP 3 C00054 BC00054  +REFP EC00054
CALL JOB:SEARCH-R1-S13D
SET P040 P006
SFTON3D P040
SMOVL C00055 BC00055 V=166.7  +MOVJ EC00055
SMOVL C00056 BC00056 V=250.0  +MOVJ EC00056
SREFP 3 C00057 BC00057  +REFP EC00057
CALL JOB:SEARCH-R1-S13D
SET P040 P006
SFTON3D P040
SMOVL C00058 BC00058 V=250.0  +MOVJ EC00058
MOVL C00059 BC00059 V=1000.0  +MOVJ EC00059 VJ=100.00
'EndPath S4328
'Path S4327
SFTOF3D
MOVJ C00060 BC00060 VJ=100.00  +MOVJ EC00060 VJ=100.00
MOVL C00061 BC00061 V=800.0  +MOVJ EC00061 VJ=100.00
SMOVL C00062 BC00062 V=166.7  +MOVJ EC00062
SREFP 3 C00063 BC00063  +REFP EC00063
CALL JOB:SEARCH-R1-S13D
SET P039 P006
SFTON3D P039
SMOVL C00064 BC00064 V=166.7  +MOVJ EC00064
SREFP 3 C00065 BC00065  +REFP EC00065
CALL JOB:SEARCH-R1-S13D
SET P039 P006
SFTON3D P039
SMOVL C00066 BC00066 V=166.7  +MOVJ EC00066
SMOVL C00067 BC00067 V=250.0  +MOVJ EC00067
SREFP 3 C00068 BC00068  +REFP EC00068
CALL JOB:SEARCH-R1-S13D
SET P039 P006
SFTON3D P039
SMOVL C00069 BC00069 V=250.0  +MOVJ EC00069
MOVL C00070 BC00070 V=1000.0  +MOVJ EC00070 VJ=100.00
'EndPath S4327
'Path S4325
SFTOF3D
MOVJ C00071 BC00071 VJ=100.00  +MOVJ EC00071 VJ=100.00
MOVL C00072 BC00072 V=666.7  +MOVJ EC00072 VJ=100.00
SMOVL C00073 BC00073 V=166.7  +MOVJ EC00073
SREFP 3 C00074 BC00074  +REFP EC00074
CALL JOB:SEARCH-R1-S13D
SET P038 P006
SFTON3D P038
SMOVL C00075 BC00075 V=166.7  +MOVJ EC00075
SREFP 3 C00076 BC00076  +REFP EC00076
CALL JOB:SEARCH-R1-S13D
SET P038 P006
SFTON3D P038
SMOVL C00077 BC00077 V=166.7  +MOVJ EC00077
SMOVL C00078 BC00078 V=166.7  +MOVJ EC00078
SMOVL C00079 BC00079 V=166.7  +MOVJ EC00079
SREFP 3 C00080 BC00080  +REFP EC00080
CALL JOB:SEARCH-R1-S13D
SET P038 P006
SFTON3D P038
SMOVL C00081 BC00081 V=166.7  +MOVJ EC00081
MOVL C00082 BC00082 V=1000.0  +MOVJ EC00082 VJ=100.00
'EndPath S4325
'Path S4324
SFTOF3D
MOVJ C00083 BC00083 VJ=100.00  +MOVJ EC00083 VJ=100.00
MOVL C00084 BC00084 V=666.7  +MOVJ EC00084 VJ=100.00
SMOVL C00085 BC00085 V=166.7  +MOVJ EC00085
SREFP 3 C00086 BC00086  +REFP EC00086
CALL JOB:SEARCH-R1-S13D
SET P037 P006
SFTON3D P037
SMOVL C00087 BC00087 V=166.7  +MOVJ EC00087
SREFP 3 C00088 BC00088  +REFP EC00088
CALL JOB:SEARCH-R1-S13D
SET P037 P006
SFTON3D P037
SMOVL C00089 BC00089 V=166.7  +MOVJ EC00089
SMOVL C00090 BC00090 V=250.0  +MOVJ EC00090
SREFP 3 C00091 BC00091  +REFP EC00091
CALL JOB:SEARCH-R1-S13D
SET P037 P006
SFTON3D P037
SMOVL C00092 BC00092 V=250.0  +MOVJ EC00092
MOVL C00093 BC00093 V=1000.0  +MOVJ EC00093 VJ=100.00
'EndPath S4324
'Path W4326
SFTOF3D
SFTON3D P037
MOVJ C00094 BC00094 VJ=100.00  +MOVJ EC00094 VJ=100.00
SMOVL C00095 BC00095 V=800.0  +MOVJ EC00095
SMOVL C00096 BC00096 V=150.0 PL=0  +MOVJ EC00096
MACRO1 MJ#(0) ARGF9
ARCON
SMOVL C00097 BC00097 V=10.0  +MOVJ EC00097
SMOVL C00098 BC00098 V=10.0  +MOVJ EC00098
ARCON
SFTON3D P038
SMOVL C00099 BC00099 V=10.0  +MOVJ EC00099
SMOVL C00100 BC00100 V=10.0  +MOVJ EC00100
SMOVL C00101 BC00101 V=10.0  +MOVJ EC00101
ARCON
SMOVL C00102 BC00102 V=10.0  +MOVJ EC00102
SMOVL C00103 BC00103 V=11.7  +MOVJ EC00103
ARCOF
SMOVL C00104 BC00104 V=800.0  +MOVJ EC00104
SMOVL C00105 BC00105 V=1000.0  +MOVJ EC00105
SFTOF3D
'EndPath W4326
MOVJ C00106 BC00106 VJ=100.00  +MOVJ EC00106 VJ=100.00
'Path W4329
SFTOF3D
SFTON3D P040
MOVJ C00107 BC00107 VJ=100.00  +MOVJ EC00107 VJ=100.00
SMOVL C00108 BC00108 V=800.0  +MOVJ EC00108
SMOVL C00109 BC00109 V=150.0 PL=0  +MOVJ EC00109
ARCON
SMOVL C00110 BC00110 V=10.0  +MOVJ EC00110
SMOVL C00111 BC00111 V=10.0  +MOVJ EC00111
SMOVL C00112 BC00112 V=10.0  +MOVJ EC00112
SMOVL C00113 BC00113 V=10.0  +MOVJ EC00113
SFTON3D P039
SMOVL C00114 BC00114 V=8.3  +MOVJ EC00114
SMOVL C00115 BC00115 V=8.3  +MOVJ EC00115
SMOVL C00116 BC00116 V=8.3  +MOVJ EC00116
ARCOF
SMOVL C00117 BC00117 V=800.0  +MOVJ EC00117
SMOVL C00118 BC00118 V=1000.0  +MOVJ EC00118
SFTOF3D
'EndPath W4329
MOVJ C00119 BC00119 VJ=100.00  +MOVJ EC00119 VJ=100.00
'Path W4330
SFTOF3D
SFTON3D P033
MOVJ C00120 BC00120 VJ=100.00  +MOVJ EC00120 VJ=100.00
SMOVL C00121 BC00121 V=800.0  +MOVJ EC00121
SMOVL C00122 BC00122 V=150.0 PL=0  +MOVJ EC00122
ARCON
SMOVL C00123 BC00123 V=10.0  +MOVJ EC00123
SMOVL C00124 BC00124 V=10.0  +MOVJ EC00124
SFTON3D P034
SMOVL C00125 BC00125 V=10.0  +MOVJ EC00125
SMOVL C00126 BC00126 V=11.7  +MOVJ EC00126
SMOVL C00127 BC00127 V=11.7  +MOVJ EC00127
SMOVL C00128 BC00128 V=11.7  +MOVJ EC00128
ARCOF
SMOVL C00129 BC00129 V=800.0  +MOVJ EC00129
SMOVL C00130 BC00130 V=1000.0  +MOVJ EC00130
SFTOF3D
'EndPath W4330
MOVJ C00131 BC00131 VJ=100.00  +MOVJ EC00131 VJ=100.00
'Path W3572
SFTOF3D
SFTON3D P036
MOVJ C00132 BC00132 VJ=100.00  +MOVJ EC00132 VJ=100.00
SMOVL C00133 BC00133 V=800.0  +MOVJ EC00133
SMOVL C00134 BC00134 V=150.0 PL=0  +MOVJ EC00134
ARCON
SMOVL C00135 BC00135 V=10.0  +MOVJ EC00135
SMOVL C00136 BC00136 V=10.0  +MOVJ EC00136
SMOVL C00137 BC00137 V=10.0  +MOVJ EC00137
SMOVL C00138 BC00138 V=10.0  +MOVJ EC00138
SFTON3D P035
SMOVL C00139 BC00139 V=8.3  +MOVJ EC00139
SMOVL C00140 BC00140 V=8.3  +MOVJ EC00140
SMOVL C00141 BC00141 V=8.3  +MOVJ EC00141
ARCOF
SMOVL C00142 BC00142 V=800.0  +MOVJ EC00142
SMOVL C00143 BC00143 V=1000.0  +MOVJ EC00143
SFTOF3D
'EndPath W3572
MOVJ C00144 BC00144 VJ=100.00  +MOVJ EC00144 VJ=100.00
MOVJ C00145 BC00145 VJ=100.00  +MOVJ EC00145 VJ=100.00
'
CALL JOB:CLEAN-R1_KM_NEW
MOVJ C00146 BC00146 VJ=100.00  +MOVJ EC00146 VJ=100.00
MOVJ C00147 BC00147 VJ=100.00  +MOVJ EC00147 VJ=100.00
MOVJ C00148 BC00148 VJ=100.00  +MOVJ EC00148 VJ=100.00
COMM PAUSE
COMM MOVJ C00149 BC00149 VJ=100.00  +MOVJ EC00149 VJ=100.00
COMM MOVL C00150 BC00150 V=800.0  +MOVJ EC00150 VJ=100.00
COMM SMOVL C00151 BC00151 V=166.7  +MOVJ EC00151
COMM SREFP 3 C00152 BC00152  +REFP EC00152
COMM CALL JOB:SEARCH-R1-S13D
COMM SET P021 P006
COMM SFTON3D P021
COMM SMOVL C00153 BC00153 V=166.7  +MOVJ EC00153
COMM SREFP 3 C00154 BC00154  +REFP EC00154
COMM CALL JOB:SEARCH-R1-S13D
COMM SET P021 P006
COMM SFTON3D P021
COMM SMOVL C00155 BC00155 V=166.7  +MOVJ EC00155
COMM SMOVL C00156 BC00156 V=250.0  +MOVJ EC00156
COMM SMOVL C00157 BC00157 V=166.7  +MOVJ EC00157
COMM SREFP 3 C00158 BC00158  +REFP EC00158
COMM CALL JOB:SEARCH-R1-S13D
COMM SET P021 P006
COMM SFTON3D P021
COMM SMOVL C00159 BC00159 V=166.7  +MOVJ EC00159
COMM MOVL C00160 BC00160 V=1000.0  +MOVJ EC00160 VJ=100.00
COMM 'EndPath S4299
COMM 'Path S4300
COMM SFTOF3D
COMM MOVJ C00161 BC00161 VJ=100.00  +MOVJ EC00161 VJ=100.00
MOVL C00162 BC00162 V=800.0  +MOVJ EC00162 VJ=100.00
SMOVL C00163 BC00163 V=166.7  +MOVJ EC00163
SREFP 3 C00164 BC00164  +REFP EC00164
CALL JOB:SEARCH-R1-S13D
SET P022 P006
SFTON3D P022
SMOVL C00165 BC00165 V=166.7  +MOVJ EC00165
SMOVL C00166 BC00166 V=166.7  +MOVJ EC00166
SREFP 3 C00167 BC00167  +REFP EC00167
CALL JOB:SEARCH-R1-S13D
SET P022 P006
SFTON3D P022
SMOVL C00168 BC00168 V=166.7  +MOVJ EC00168
SMOVL C00169 BC00169 V=250.0  +MOVJ EC00169
SMOVL C00170 BC00170 V=166.7  +MOVJ EC00170
SREFP 3 C00171 BC00171  +REFP EC00171
CALL JOB:SEARCH-R1-S13D
SET P022 P006
SFTON3D P022
SMOVL C00172 BC00172 V=166.7  +MOVJ EC00172
MOVL C00173 BC00173 V=1000.0  +MOVJ EC00173 VJ=100.00
'EndPath S4300
'Path S4301
SFTOF3D
MOVJ C00174 BC00174 VJ=100.00  +MOVJ EC00174 VJ=100.00
MOVL C00175 BC00175 V=800.0  +MOVJ EC00175 VJ=100.00
SMOVL C00176 BC00176 V=166.7  +MOVJ EC00176
SREFP 3 C00177 BC00177  +REFP EC00177
CALL JOB:SEARCH-R1-S13D
SET P023 P006
SFTON3D P023
SMOVL C00178 BC00178 V=166.7  +MOVJ EC00178
SREFP 3 C00179 BC00179  +REFP EC00179
CALL JOB:SEARCH-R1-S13D
SET P023 P006
SFTON3D P023
SMOVL C00180 BC00180 V=166.7  +MOVJ EC00180
MOVL C00181 BC00181 V=1000.0  +MOVJ EC00181 VJ=100.00
'EndPath S4301
'Path S4302
SFTOF3D
MOVJ C00182 BC00182 VJ=100.00  +MOVJ EC00182 VJ=100.00
MOVL C00183 BC00183 V=800.0  +MOVJ EC00183 VJ=100.00
SMOVL C00184 BC00184 V=166.7  +MOVJ EC00184
SREFP 3 C00185 BC00185  +REFP EC00185
CALL JOB:SEARCH-R1-S13D
SET P024 P006
SFTON3D P024
SMOVL C00186 BC00186 V=166.7  +MOVJ EC00186
SREFP 3 C00187 BC00187  +REFP EC00187
CALL JOB:SEARCH-R1-S13D
SET P024 P006
SFTON3D P024
SMOVL C00188 BC00188 V=166.7  +MOVJ EC00188
MOVL C00189 BC00189 V=1000.0  +MOVJ EC00189 VJ=100.00
'EndPath S4302
'Path S4303
SFTOF3D
MOVJ C00190 BC00190 VJ=100.00  +MOVJ EC00190 VJ=100.00
MOVL C00191 BC00191 V=800.0  +MOVJ EC00191 VJ=100.00
SMOVL C00192 BC00192 V=166.7  +MOVJ EC00192
SREFP 3 C00193 BC00193  +REFP EC00193
CALL JOB:SEARCH-R1-S13D
SET P025 P006
SFTON3D P025
SMOVL C00194 BC00194 V=166.7  +MOVJ EC00194
SREFP 3 C00195 BC00195  +REFP EC00195
CALL JOB:SEARCH-R1-S13D
SET P025 P006
SFTON3D P025
SMOVL C00196 BC00196 V=166.7  +MOVJ EC00196
MOVL C00197 BC00197 V=1000.0  +MOVJ EC00197 VJ=100.00
'EndPath S4303
'Path S4313
SFTOF3D
MOVJ C00198 BC00198 VJ=100.00  +MOVJ EC00198 VJ=100.00
MOVL C00199 BC00199 V=800.0  +MOVJ EC00199 VJ=100.00
SMOVL C00200 BC00200 V=166.7  +MOVJ EC00200
SREFP 3 C00201 BC00201  +REFP EC00201
CALL JOB:SEARCH-R1-S13D
SET P032 P006
SFTON3D P032
SMOVL C00202 BC00202 V=166.7  +MOVJ EC00202
SREFP 3 C00203 BC00203  +REFP EC00203
CALL JOB:SEARCH-R1-S13D
SET P032 P006
SFTON3D P032
SMOVL C00204 BC00204 V=166.7  +MOVJ EC00204
SMOVL C00205 BC00205 V=250.0  +MOVJ EC00205
SMOVL C00206 BC00206 V=166.7  +MOVJ EC00206
SREFP 3 C00207 BC00207  +REFP EC00207
CALL JOB:SEARCH-R1-S13D
SET P032 P006
SFTON3D P032
SMOVL C00208 BC00208 V=166.7  +MOVJ EC00208
MOVL C00209 BC00209 V=1000.0  +MOVJ EC00209 VJ=100.00
'EndPath S4313
'Path S4312
SFTOF3D
MOVJ C00210 BC00210 VJ=100.00  +MOVJ EC00210 VJ=100.00
COMM PAUSE
COMM MOVL C00211 BC00211 V=800.0  +MOVJ EC00211 VJ=100.00
COMM SMOVL C00212 BC00212 V=166.7  +MOVJ EC00212
COMM SREFP 3 C00213 BC00213  +REFP EC00213
COMM CALL JOB:SEARCH-R1-S13D
COMM SET P031 P006
COMM SFTON3D P031
COMM SMOVL C00214 BC00214 V=166.7  +MOVJ EC00214
COMM SREFP 3 C00215 BC00215  +REFP EC00215
COMM CALL JOB:SEARCH-R1-S13D
COMM SET P031 P006
COMM SFTON3D P031
COMM SMOVL C00216 BC00216 V=166.7  +MOVJ EC00216
COMM SMOVL C00217 BC00217 V=250.0  +MOVJ EC00217
COMM SMOVL C00218 BC00218 V=166.7  +MOVJ EC00218
COMM SREFP 3 C00219 BC00219  +REFP EC00219
COMM CALL JOB:SEARCH-R1-S13D
COMM SET P031 P006
COMM SFTON3D P031
COMM SMOVL C00220 BC00220 V=250.0  +MOVJ EC00220
COMM MOVL C00221 BC00221 V=1000.0  +MOVJ EC00221 VJ=100.00
COMM 'EndPath S4312
COMM 'Path W4314
COMM SFTOF3D
COMM SFTON3D P031
COMM MOVJ C00222 BC00222 VJ=100.00  +MOVJ EC00222 VJ=100.00
COMM SMOVL C00223 BC00223 V=800.0  +MOVJ EC00223
COMM SMOVL C00224 BC00224 V=150.0 PL=0  +MOVJ EC00224
COMM MACRO1 MJ#(0) ARGF14
COMM ARCON
COMM SMOVL C00225 BC00225 V=11.7  +MOVJ EC00225
COMM SMOVL C00226 BC00226 V=11.7  +MOVJ EC00226
COMM ARCON
COMM SMOVL C00227 BC00227 V=11.7  +MOVJ EC00227
COMM ARCOF
COMM SMOVL C00228 BC00228 V=800.0  +MOVJ EC00228
COMM SMOVL C00229 BC00229 V=1000.0  +MOVJ EC00229
COMM SFTOF3D
COMM 'EndPath W4314
COMM 'Path W4315
COMM SFTOF3D
COMM SFTON3D P031
COMM MOVJ C00230 BC00230 VJ=100.00  +MOVJ EC00230 VJ=100.00
COMM SMOVL C00231 BC00231 V=800.0  +MOVJ EC00231
COMM SMOVL C00232 BC00232 V=150.0 PL=0  +MOVJ EC00232
COMM MACRO1 MJ#(0) ARGF6
COMM ARCON
COMM SMOVL C00233 BC00233 V=10.8  +MOVJ EC00233
COMM SMOVL C00234 BC00234 V=10.8  +MOVJ EC00234
COMM SMOVL C00235 BC00235 V=10.0  +MOVJ EC00235
COMM SMOVL C00236 BC00236 V=10.0  +MOVJ EC00236
COMM ARCOF
COMM SMOVL C00237 BC00237 V=800.0  +MOVJ EC00237
COMM SMOVL C00238 BC00238 V=333.3  +MOVJ EC00238
COMM SMOVL C00239 BC00239 V=133.3  +MOVJ EC00239
COMM ARCON
COMM SMOVL C00240 BC00240 V=11.7  +MOVJ EC00240
COMM SMOVL C00241 BC00241 V=11.7  +MOVJ EC00241
COMM ARCOF
COMM SMOVL C00242 BC00242 V=250.0  +MOVJ EC00242
COMM SMOVL C00243 BC00243 V=1000.0  +MOVJ EC00243
COMM SFTOF3D
COMM 'EndPath W4315
MOVJ C00244 BC00244 VJ=100.00  +MOVJ EC00244 VJ=100.00
'
'Path W4316
SFTOF3D
SFTON3D P032
MOVJ C00245 BC00245 VJ=100.00  +MOVJ EC00245 VJ=100.00
SMOVL C00246 BC00246 V=800.0  +MOVJ EC00246
SMOVL C00247 BC00247 V=150.0 PL=0  +MOVJ EC00247
MACRO1 MJ#(0) ARGF21
ARCON
SMOVL C00248 BC00248 V=10.0  +MOVJ EC00248
SMOVL C00249 BC00249 V=10.0  +MOVJ EC00249
SMOVL C00250 BC00250 V=8.3  +MOVJ EC00250
ARCON
SMOVL C00251 BC00251 V=9.2  +MOVJ EC00251
SMOVL C00252 BC00252 V=9.2  +MOVJ EC00252
ARCOF
SMOVL C00253 BC00253 V=800.0  +MOVJ EC00253
SMOVL C00254 BC00254 V=1000.0  +MOVJ EC00254
SFTOF3D
'EndPath W4316
MOVJ C00255 BC00255 VJ=100.00  +MOVJ EC00255 VJ=100.00
MOVJ C00256 BC00256 VJ=100.00  +MOVJ EC00256 VJ=100.00
MOVJ C00257 BC00257 VJ=100.00  +MOVJ EC00257 VJ=100.00
'Path W4317
SFTOF3D
SFTON3D P032
MOVJ C00258 BC00258 VJ=100.00  +MOVJ EC00258 VJ=100.00
SMOVL C00259 BC00259 V=800.0  +MOVJ EC00259
SMOVL C00260 BC00260 V=150.0 PL=0  +MOVJ EC00260
ARCON
SMOVL C00261 BC00261 V=10.0  +MOVJ EC00261
SMOVL C00262 BC00262 V=10.0  +MOVJ EC00262
SMOVL C00263 BC00263 V=10.0  +MOVJ EC00263
ARCON
SMOVL C00264 BC00264 V=10.0  +MOVJ EC00264
ARCOF
SMOVL C00265 BC00265 V=800.0  +MOVJ EC00265
SMOVL C00266 BC00266 V=1000.0  +MOVJ EC00266
SFTOF3D
'EndPath W4317
MOVJ C00267 BC00267 VJ=100.00  +MOVJ EC00267 VJ=100.00
'Path W4318
SFTOF3D
SFTON3D P032
MOVJ C00268 BC00268 VJ=100.00  +MOVJ EC00268 VJ=100.00
SMOVL C00269 BC00269 V=800.0  +MOVJ EC00269
SMOVL C00270 BC00270 V=150.0 PL=0  +MOVJ EC00270
SWVON WEV#(99)
MACRO1 MJ#(0) ARGF9
ARCON
SMOVL C00271 BC00271 V=9.2  +MOVJ EC00271
ARCOF
SWVOF
SMOVL C00272 BC00272 V=33.3  +MOVJ EC00272
TIMER T=2.00
ARCON
TIMER T=0.50
SMOVL C00273 BC00273 V=8.3  +MOVJ EC00273
ARCOF
SMOVL C00274 BC00274 V=800.0  +MOVJ EC00274
SFTOF3D
'EndPath W4318
MOVJ C00275 BC00275 VJ=100.00  +MOVJ EC00275 VJ=100.00
'
'Path W4310
SFTOF3D
SFTON3D P024
MOVJ C00276 BC00276 VJ=100.00  +MOVJ EC00276 VJ=100.00
SMOVL C00277 BC00277 V=800.0  +MOVJ EC00277
SMOVL C00278 BC00278 V=150.0 PL=0  +MOVJ EC00278
MACRO1 MJ#(0) ARGF14
ARCON
SWVON WEV#(22)
SMOVL C00279 BC00279 V=10.0  +MOVJ EC00279
SFTON3D P025
SMOVL C00280 BC00280 V=10.0  +MOVJ EC00280
SMOVL C00281 BC00281 V=10.0  +MOVJ EC00281
ARCOF
SWVOF
SMOVL C00282 BC00282 V=800.0  +MOVJ EC00282
SMOVL C00283 BC00283 V=1000.0  +MOVJ EC00283
SFTOF3D
'EndPath W4310
'Path W4311
SFTOF3D
SFTON3D P024
MOVJ C00284 BC00284 VJ=100.00  +MOVJ EC00284 VJ=100.00
SMOVL C00285 BC00285 V=800.0  +MOVJ EC00285
SMOVL C00286 BC00286 V=150.0 PL=0  +MOVJ EC00286
ARCON
SWVON WEV#(22)
SMOVL C00287 BC00287 V=10.0  +MOVJ EC00287
SFTON3D P023
SMOVL C00288 BC00288 V=10.0  +MOVJ EC00288
SMOVL C00289 BC00289 V=10.0  +MOVJ EC00289
ARCOF
SWVOF
SMOVL C00290 BC00290 V=800.0  +MOVJ EC00290
SMOVL C00291 BC00291 V=1000.0  +MOVJ EC00291
SFTOF3D
'EndPath W4311
'
MOVJ C00292 BC00292 VJ=100.00  +MOVJ EC00292 VJ=100.00
MOVJ C00293 BC00293 VJ=100.00  +MOVJ EC00293 VJ=100.00
MOVJ C00294 BC00294 VJ=100.00  +MOVJ EC00294 VJ=100.00
'Path W4331
SFTOF3D
SFTON3D P022
MOVJ C00295 BC00295 VJ=100.00  +MOVJ EC00295 VJ=100.00
SMOVL C00296 BC00296 V=800.0  +MOVJ EC00296
SMOVL C00297 BC00297 V=150.0 PL=0  +MOVJ EC00297
MACRO1 MJ#(0) ARGF21
ARCON
SMOVL C00298 BC00298 V=9.2  +MOVJ EC00298
SMOVL C00299 BC00299 V=9.2  +MOVJ EC00299
SMOVL C00300 BC00300 V=9.2  +MOVJ EC00300
SMOVL C00301 BC00301 V=9.2  +MOVJ EC00301
SMOVL C00302 BC00302 V=9.2  +MOVJ EC00302
SMOVL C00303 BC00303 V=9.2  +MOVJ EC00303
ARCOF
SFTOF3D
SMOVL C00304 BC00304 V=800.0  +MOVJ EC00304
SMOVL C00305 BC00305 V=333.3  +MOVJ EC00305
SFTOF3D
'EndPath W4331
MOVJ C00306 BC00306 VJ=100.00  +MOVJ EC00306 VJ=100.00
MOVJ C00307 BC00307 VJ=100.00  +MOVJ EC00307 VJ=100.00
'Path W4306
SFTOF3D
SFTON3D P022
MOVJ C00308 BC00308 VJ=100.00  +MOVJ EC00308 VJ=100.00
SMOVL C00309 BC00309 V=800.0  +MOVJ EC00309
SMOVL C00310 BC00310 V=150.0 PL=0  +MOVJ EC00310
ARCON
SMOVL C00311 BC00311 V=10.0  +MOVJ EC00311
SMOVL C00312 BC00312 V=10.0  +MOVJ EC00312
SMOVL C00313 BC00313 V=10.0  +MOVJ EC00313
SMOVL C00314 BC00314 V=10.0  +MOVJ EC00314
SMOVL C00315 BC00315 V=10.0  +MOVJ EC00315
ARCOF
SMOVL C00316 BC00316 V=800.0  +MOVJ EC00316
SMOVL C00317 BC00317 V=1000.0  +MOVJ EC00317
SFTOF3D
'EndPath W4306
MOVJ C00318 BC00318 VJ=100.00  +MOVJ EC00318 VJ=100.00
'Path W4332
SFTOF3D
SFTON3D P022
MOVJ C00319 BC00319 VJ=100.00  +MOVJ EC00319 VJ=100.00
SMOVL C00320 BC00320 V=800.0  +MOVJ EC00320
SMOVL C00321 BC00321 V=150.0 PL=0  +MOVJ EC00321
SMOVL C00322 BC00322 V=9.2  +MOVJ EC00322
MACRO1 MJ#(0) ARGF9
ARCON
SWVON WEV#(99)
SMOVL C00323 BC00323 V=9.2  +MOVJ EC00323
ARCOF
SWVOF
SMOVL C00324 BC00324 V=9.2  +MOVJ EC00324
TIMER T=3.00
ARCON
SMOVL C00325 BC00325 V=9.2  +MOVJ EC00325
ARCOF
SMOVL C00326 BC00326 V=800.0  +MOVJ EC00326
SFTOF3D
'EndPath W4332
'
MOVJ C00327 BC00327 VJ=100.00  +MOVJ EC00327 VJ=100.00
COMM PAUSE
COMM 'Path W4304
COMM SFTOF3D
COMM SFTON3D P021
COMM MOVJ C00328 BC00328 VJ=100.00  +MOVJ EC00328 VJ=100.00
COMM SMOVL C00329 BC00329 V=800.0  +MOVJ EC00329
COMM SMOVL C00330 BC00330 V=150.0 PL=0  +MOVJ EC00330
COMM MACRO1 MJ#(0) ARGF14
COMM ARCON
COMM SMOVL C00331 BC00331 V=10.0  +MOVJ EC00331
COMM SMOVL C00332 BC00332 V=10.0  +MOVJ EC00332
COMM SMOVL C00333 BC00333 V=10.0  +MOVJ EC00333
COMM ARCOF
COMM SMOVL C00334 BC00334 V=800.0  +MOVJ EC00334
COMM SMOVL C00335 BC00335 V=1000.0  +MOVJ EC00335
COMM SFTOF3D
COMM 'EndPath W4304
COMM 'Path W4305
COMM SFTOF3D
COMM SFTON3D P021
COMM MOVJ C00336 BC00336 VJ=100.00  +MOVJ EC00336 VJ=100.00
COMM SMOVL C00337 BC00337 V=800.0  +MOVJ EC00337
COMM SMOVL C00338 BC00338 V=150.0 PL=0  +MOVJ EC00338
COMM MACRO1 MJ#(0) ARGF6
COMM ARCON
COMM SMOVL C00339 BC00339 V=10.8  +MOVJ EC00339
COMM SMOVL C00340 BC00340 V=10.8  +MOVJ EC00340
COMM SMOVL C00341 BC00341 V=10.8  +MOVJ EC00341
COMM SMOVL C00342 BC00342 V=11.7  +MOVJ EC00342
COMM ARCOF
COMM SMOVL C00343 BC00343 V=800.0  +MOVJ EC00343
COMM SMOVL C00344 BC00344 V=333.3  +MOVJ EC00344
COMM SMOVL C00345 BC00345 V=333.3  +MOVJ EC00345
COMM ARCON
COMM SMOVL C00346 BC00346 V=11.7  +MOVJ EC00346
COMM ARCOF
COMM SMOVL C00347 BC00347 V=333.3  +MOVJ EC00347
COMM SMOVL C00348 BC00348 V=1000.0  +MOVJ EC00348
COMM SFTOF3D
COMM 'EndPath W4305
MOVJ C00349 BC00349 VJ=100.00  +MOVJ EC00349 VJ=100.00
MOVJ C00350 BC00350 VJ=100.00  +MOVJ EC00350 VJ=100.00
MOVJ C00351 BC00351 VJ=100.00  +MOVJ EC00351 VJ=100.00
END
